PROGRAM POU_1
VAR
	
	objectDetected : BOOL := FALSE;

	blackObject : BOOL := FALSE;	
	redObject : BOOL := FALSE;
	
	motorOn : BOOL := FALSE;
	actuatorMove : BOOL := FALSE;
	
	objectSorted : BOOL := FALSE;
	
	startTimer : BOOL := FALSE;
	TON_0 : TON;	

END_VAR

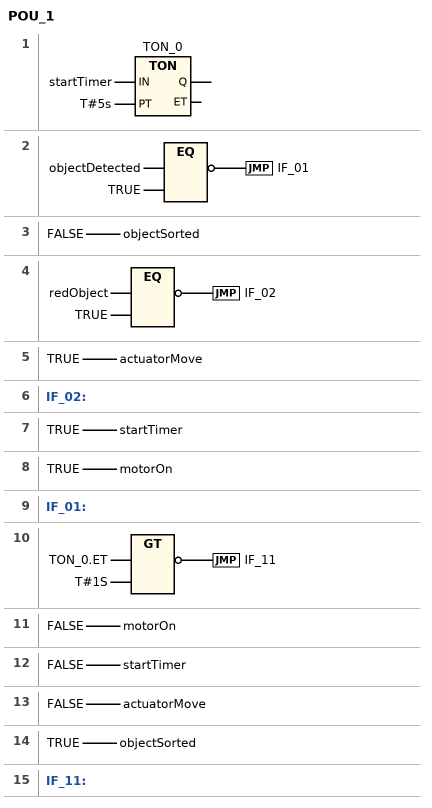
// NETWORK 1
TON_0(IN := startTimer, PT := T#5s); // TON

// NETWORK 2
IF NOT (objectDetected = TRUE) THEN JMP IF_01; END_IF

// NETWORK 3
objectSorted := FALSE;

// NETWORK 4
IF NOT (redObject = TRUE) THEN JMP IF_02; END_IF

// NETWORK 5
actuatorMove := TRUE;

// NETWORK 6
IF_02: ;

// NETWORK 7
startTimer := TRUE;

// NETWORK 8
motorOn := TRUE;

// NETWORK 9
IF_01: ;

// NETWORK 10
IF NOT (TON_0.ET > T#1S) THEN JMP IF_11; END_IF

// NETWORK 11
motorOn := FALSE;

// NETWORK 12
startTimer := FALSE;

// NETWORK 13
actuatorMove := FALSE;

// NETWORK 14
objectSorted := TRUE;

// NETWORK 15
IF_11: ;

END_PROGRAM

(* stored: Version 1.1.0.1, ProductVersion 3.1.4024.3
   POU POU_1: Id {3c72f77c-2748-4769-8897-b2b3884e4a37}, SpecialFunc None *)
